Fanuc TP program (LS listing): OPEN_GRIPPER.LS

/PROG  OPEN_GRIPPER
/ATTR
OWNER		= MNEDITOR;
COMMENT		= "";
PROG_SIZE	= 160;
CREATE		= DATE 22-10-07  TIME 07:17:04;
MODIFIED	= DATE 22-10-07  TIME 13:04:18;
FILE_NAME	= ;
VERSION		= 0;
LINE_COUNT	= 2;
MEMORY_SIZE	= 524;
PROTECT		= READ_WRITE;
TCD:  STACK_SIZE	= 0,
      TASK_PRIORITY	= 50,
      TIME_SLICE	= 0,
      BUSY_LAMP_OFF	= 0,
      ABORT_REQUEST	= 0,
      PAUSE_REQUEST	= 0;
DEFAULT_GROUP	= *,*,*,*,*;
CONTROL_CODE	= 00000000 00000000;
/APPL
/MN
   1:  DO[9]=ON ;
   2:  DO[10]=OFF ;
/POS
/END
